(* PLC project CoDeSys External Library Template, WAGO e!COCKPIT e!COCKPIT, author 3S - Smart Software Solutions GmbH *)
(* stored: creationDateTime 2019-10-29T12:22:40.8971617, version 3.5.5.30, modificationDateTime 2019-10-24T14:40:07.960949, organization 3S - Smart Software Solutions GmbH *)
(* Library project template with all possible element types, docu and a sample project structure *)

FUNCTION fnKomunikatInOutZeruj : BOOL
  VAR_IN_OUT
    typKomunikat : typKomunikat;
  END_VAR

            typKomunikat.sZnacznik := '';
typKomunikat.sTypKomunikatu := '';
typKomunikat.sMnemonikWlasciciela := '';
typKomunikat.sMnemonikWlascicielaExt := '';
typKomunikat.sMACAdres := '';
typKomunikat.sIDZrodla := '';
typKomunikat.sIDZrodlaLokalizacja := '';
typKomunikat.sIDZrodlaUrzadzenie := '';
typKomunikat.sIDPrzeznaczenia :='' ;
typKomunikat.sIDPrzeznaczeniaLokalizacja := '';
typKomunikat.sIDPrzeznaczeniaUrzadzenie := '';
typKomunikat.sDlugoscPolaDanych := '';
typKomunikat.sMarkerCzasowy := '';
typKomunikat.sRezerwa := '';
typKomunikat.sDane := '';
          
END_FUNCTION
